Staubli VAL3: CompareStrArray.pgx

public program CompareStrArray(string& x_sFirst[] (dimensions=1), string& x_sSecond[] (dimensions=1), bool& x_bRes (dimensions=1))
  local num l_i
begin
  //比较两个字符串数组是否相等
  //相等返回x_bRes=true,否则x_bRes=false

  x_bRes=false
  //维数不等
  if size(x_sFirst)!=size(x_sSecond)
    return
  endIf
  //
  l_i=0
  for l_i=0 to size(x_sFirst)-1
    if x_sFirst[l_i]!=x_sSecond[l_i]
      return
    endIf
  endFor
  x_bRes=true
end
